# EPICS autosave request: motorApp/Db/basic_asyn_motor_settings.req
# FILE... motor_settings.req

file basic_motor_settings.req P=$(P),M=$(M)
